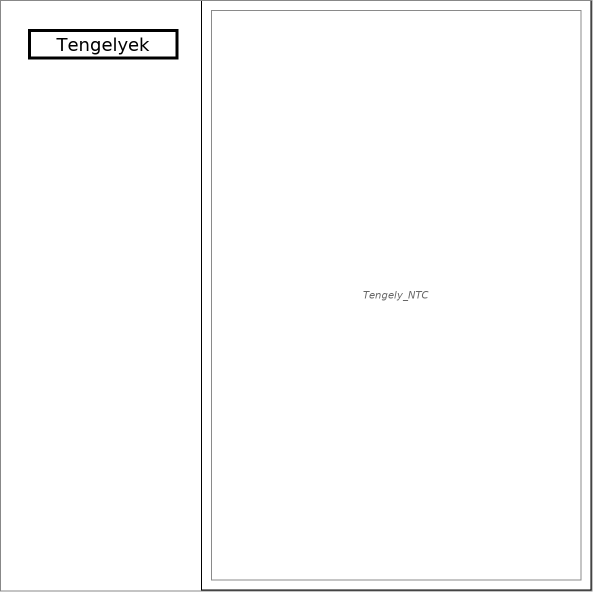
VISUALIZATION Tengelyek  // 593x592
    Group (201,0 390x590)
        Rectangle (0,0 390x590)
        TabControl (10,10 370x570)
            shows Tengely_NTC()
            shows Tengely_Pt1000()
            [0]: TabTitle=NTC oldal
            [1]: TabTitle=Pt1000 oldal
    RoundedRectangle (28,29 150x30)
    Label (28,30 150x30), "Tengelyek"
END_VISUALIZATION

(* stored: Version 1.1.0.1, ProductVersion 3.1.4024.11
   Visu Tengelyek: Id {cdec7216-f6be-4bb8-9927-496a113037b9} *)
